// TIA Portal V20 export
TYPE "typeHmiParameterParameters"
// stored: Access Published, Namespace Unit1
   STRUCT
      "Bool" { S7_SetPoint := 'True'} : Array[0..100] of Bool;
      Data { S7_SetPoint := 'True'} : Array[0..100] of LReal;
   END_STRUCT;
END_TYPE
